FUNCTION_BLOCK Seq_Ausrichten EXTENDS FB_Basis IMPLEMENTS I_Sequenz
VAR_INPUT
	// Skillzuweisung
	R_Move					:I_Skill_RoboterErweitert;
	
	// Prozessparameter		
	RobParam				:ARRAY[0..1] OF sRoboterProzessVariablen;
	ErreichtParam			:sKraftVariablen;
END_VAR
VAR_OUTPUT
END_VAR
VAR
	ErreichtParamReset		:sKraftVariablen;
	Counter			:INT;
END_VAR

// Ablauf
ACT_Ablauf();

// Zustandshandling
CASE iState OF
	0:	// BEREIT
		IF bStart THEN
			iState := 1;
		END_IF
	1:	// LAUFEND
		IF eSysCommand = 4 THEN
			bReset := TRUE;
			SFCReset := TRUE;
		END_IF
		
		IF bBeendet OR bReset THEN
			bReset := FALSE;
			SFCReset := FALSE;
			iState := 0;
		END_IF
	2: // ABGESCHLOSSEN
		IF SFCCurrentStep = 'Init' THEN
			iState := 0;
		END_IF
END_CASE

ACTION ACT_Ablauf:
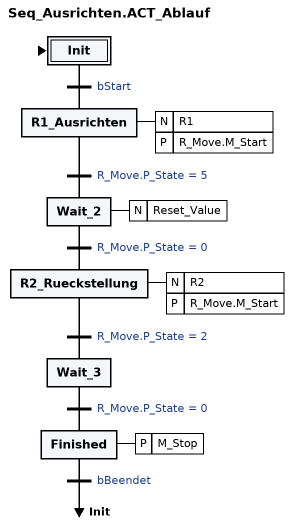
INITIAL_STEP Init:
END_STEP
TRANSITION FROM Init TO R1_Ausrichten
    := bStart;
END_TRANSITION
STEP R1_Ausrichten:
    R1(N);
    R_Move.M_Start(P);
END_STEP
TRANSITION FROM R1_Ausrichten TO Wait_2
    := R_Move.P_State = 5;
END_TRANSITION
STEP Wait_2:
    Reset_Value(N);
END_STEP
TRANSITION FROM Wait_2 TO R2_Rueckstellung
    := R_Move.P_State = 0;
END_TRANSITION
STEP R2_Rueckstellung:
    R2(N);
    R_Move.M_Start(P);
END_STEP
TRANSITION FROM R2_Rueckstellung TO Wait_3
    := R_Move.P_State = 2;
END_TRANSITION
STEP Wait_3:
END_STEP
TRANSITION FROM Wait_3 TO Finished
    := R_Move.P_State = 0;
END_TRANSITION
STEP Finished:
    M_Stop(P);
END_STEP
TRANSITION FROM Finished TO Init
    := bBeendet;
END_TRANSITION
END_ACTION

ACTION R1:
R_Move.P_RobotParam := RobParam[0];
R_Move.P_Erreicht := ErreichtParam;
END_ACTION

ACTION R2:
R_Move.P_RobotParam := RobParam[1];
END_ACTION

ACTION Reset_Value:
ErreichtParamReset.Fx := 0;
ErreichtParamReset.Fy := 0;
ErreichtParamReset.Fz := 0;

R_Move.P_Erreicht := ErreichtParamReset;
END_ACTION

END_FUNCTION_BLOCK

(* stored: Version 1.1.0.1
   POU Seq_Ausrichten: Id {11c37351-4bb3-48e4-a5a4-7c8c23eef462}, SpecialFunc None
   Folder 01_Zuweisung: Id {78d1a69a-9902-4c80-a12a-f642d1fb3a8a}
   Action ACT_Ablauf: Id {930c26a3-764f-4680-a200-e8adba9093be}
   Action R1: Id {d5218329-08e3-46e2-98f2-8142e2c2e2aa}
   Action R2: Id {95b8ba9e-adaf-43f6-bd71-5982c734e379}
   Action Reset_Value: Id {2af7a2d4-36e5-40f7-9113-6606e7c01c3b} *)
